TYPE FromXMC2ToMainControl :
STRUCT
	EM_origE_DistanceLevitationFiltered	: REAL;
	EM_origE_DistanceGuidanceFiltered	: REAL;
	EM_origE_DistanceRawLev11			: REAL;
	EM_origE_DistanceRawLev12			: REAL;
	EM_origE_DistanceRawLev21			: REAL;
	EM_origE_DistanceRawLev22			: REAL;
	EM_origE_DistanceRawGuid11			: REAL;
	EM_origE_DistanceRawGuid12			: REAL;
	EM_origE_IMUX						: REAL;
	EM_origE_IMUY						: REAL;
	EM_origE_IMUZ						: REAL;
	EM_origE_VelocityZFiltered			: REAL;
	EM_origE_TemperatureBox				: REAL;
	EM_origE_TemperatureLev0			: REAL;
	EM_origE_TemperatureLev1			: REAL;
	EM_origE_TemperatureGuid			: REAL;
	EM_origE_PressureBox				: REAL;
	EM_origE_CurrentLev					: REAL;
	EM_origE_CurrentGuid				: REAL;
	
	EM_origE_SafetyCounter				: UDINT;
	EM_origE_State						: USINT;
	EM_origE_WarnBits					: ARRAY [0..10] OF UDINT;
	EM_origE_ErrBits					: ARRAY [0..10] OF UDINT;
	EM_origE_Timestamp					: UDINT;
	
	EM_origE_LoggingCounterIn			: USINT;
	EM_origE_LoggingCounterSize			: USINT;
	EM_origE_LoggingCounterBuf			: ARRAY [0..9] OF BYTE;
END_STRUCT
END_TYPE

(* stored: Version 1.1.0.1, ProductVersion 3.1.4024.12
   DUT FromXMC2ToMainControl: Id {fd5d9cde-a5db-4c32-8e12-66824652bfa3} *)
